PROGRAM Main
VAR
END_VAR

END_PROGRAM

(* stored: Version 1.1.0.1, ProductVersion 3.1.4024.3
   POU Main: Id {4ac9dfbf-8341-45a8-a94d-1a4b17e4330e}, SpecialFunc None *)
